(* CoDeSys 2.3 export: LEVEL.EXP *)

(* Data type *)
TYPE Level :
(
    BathTop,
    BathMiddle,
    BathLower,
    TankTop,
    TankMiddle,
    TankLower,
    USBlock,
    USBlockTop,
    WarmBlock,
    PumpBlock,
    BarbBlock,
    SkimerBlock,
    FillBathStop
);
END_TYPE
